PROGRAM prgHouse
VAR
	fbHouse				: FB_HouseC_Power_Virtual;
	bHouseEnabled		: BOOL;						//{#lynus.ag#()}
	lrPowerHouse		: LREAL;					//{#lynus.ag#()}
	lrPowerHouseCaluclated: LREAL;					//{#lynus.ag#()}
END_VAR
VAR PERSISTENT
	bEnableHouse		: BOOL:=true;						//{#lynus.ag#()}
END_VAR


fbHouse(
	bEnable:= bEnableHouse, 
	diNrOfEMS_IN:= , //prgEMS.fbEMS.diNrOfEMS_OUT, 
	bSetDefault:= , 
	lrCounterConsumptionSetDefault:= , 
	lrCounterProductionSetDefault:= , 
	stDataHouseC=> , 
	diNrOfHouseC_OUT=> );

bHouseEnabled := fbHouse.stDataHouseC.bEnabled;
lrPowerHouse := fbHouse.stDataHouseC.lrPower;	
	
lrPowerHouseCaluclated := prgBattery.lrPowerBattery + prgPV.lrPowerPV + prgGrid.lrPowerGrid;

END_PROGRAM

(* stored: Version 1.1.0.1, ProductVersion 3.1.4024.12
   POU prgHouse: Id {1004e12f-88fd-4838-a3c1-f7a079c901cf}, SpecialFunc None *)
